% RSLogix 500 project PLC_1_EXAM_1.RSS, saved by version 12.00.00.00 %
PROJECT "UNTITLED"    % processor: Bul.1763 MicroLogix 1100 Series B %

PROGRAM FILES
  LAD 2   5 rungs

DATA FILES
  O0 OUTPUT  5 elements
  I1 INPUT  6 elements
  S2 STATUS  66 elements
  B3 BINARY  1 elements
  T4 TIMER  1 elements
  C5 COUNTER  1 elements
  R6 CONTROL  1 elements
  N7 INTEGER  1 elements
  F8 FLOAT  1 elements

LADDER 2
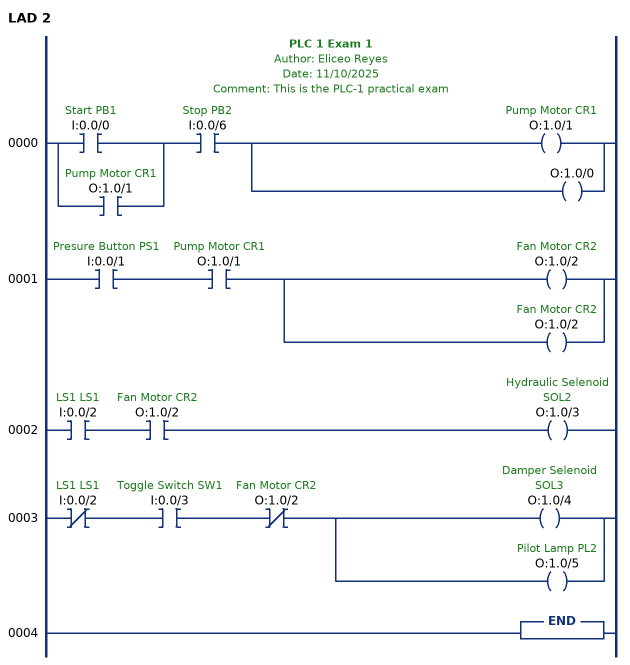
% Rung: 0 %
% TITLE: PLC 1 Exam 1 %
% Author: Eliceo Reyes
% Date: 11/10/2025
% Comment: This is the PLC-1 practical exam %
SOR BST XIC I:0.0/0 NXB XIC O:1.0/1 BND XIC I:0.0/6 BST OTE O:1.0/1 NXB OTE O:1.0/0 BND EOR
%   I:0.0/0  PB1  "Start" %
%   O:1.0/1  CR1  "Pump Motor" %
%   I:0.0/6  PB2  "Stop" %
% Rung: 1 %
SOR XIC I:0.0/1 XIC O:1.0/1 BST OTE O:1.0/2 NXB OTE O:1.0/2 BND EOR
%   I:0.0/1  PS1  "Presure Button" %
%   O:1.0/1  CR1  "Pump Motor" %
%   O:1.0/2  CR2  "Fan Motor" %
% Rung: 2 %
SOR XIC I:0.0/2 XIC O:1.0/2 OTE O:1.0/3 EOR
%   I:0.0/2  LS1  "LS1" %
%   O:1.0/2  CR2  "Fan Motor" %
%   O:1.0/3  SOL2  "Hydraulic Selenoid" %
% Rung: 3 %
SOR XIO I:0.0/2 XIC I:0.0/3 XIO O:1.0/2 BST OTE O:1.0/4 NXB OTE O:1.0/5 BND EOR
%   I:0.0/2  LS1  "LS1" %
%   I:0.0/3  SW1  "Toggle Switch" %
%   O:1.0/2  CR2  "Fan Motor" %
%   O:1.0/4  SOL3  "Damper Selenoid" %
%   O:1.0/5  PL2  "Pilot Lamp" %
% Rung: 4 %
SOR END EOR

OTHER DOCUMENTED ADDRESSES
  O:0.0/0  PM  "Pump Motor"
  O:0.0/1  PL1  "Pilot Lamp"
  O:0.0/2  SOL1  "Pneumatic"
